// TIA Portal V20 export
DATA_BLOCK "OPERATOR_PROMPT_DB"   // DB86
{ S7_Optimized_Access := 'TRUE' }
AUTHOR : Tesla
FAMILY : OperatorPrompt
// stored: MemoryReserve 100
   VAR
      "IF" { ExternalAccessible := 'False'; ExternalVisible := 'False'; ExternalWritable := 'False'; S7_SetPoint := 'True'} : "OPERATOR_PROMPT_UDT";
   END_VAR
BEGIN
END_DATA_BLOCK
